// TIA Portal V18 export
DATA_BLOCK "Flowrate"   // DB205
{ S7_Optimized_Access := 'TRUE' }
VERSION : 0.1
// stored: AutoNumber true, DBAccessibleFromOPCUA true, IsOnlyStoredInLoadMemory false, IsRetainMemResEnabled false, IsWriteProtectedInAS false, MemoryReserve 100
   VAR
      Current : Struct
         "A" : Real;
         "B" : Real;
         Mixed : Real;
      END_STRUCT;
      "current in ml/min" : Struct
         "A" : Real;
         "B" : Real;
         Mixed : Real;
      END_STRUCT;
      "current in L/min" : Struct
         "A" : Real;
         "B" : Real;
         Mixed : Real;
      END_STRUCT;
      "current in KG/min" : Struct
         "A" : Real;
         "B" : Real;
         Mixed : Real;
      END_STRUCT;
      "Volume in ml" : Struct
         "A" : Real;
         "B" : Real;
         mixed : Real;
      END_STRUCT;
      "Volume in L" : Struct
         "A" : Real;
         "B" : Real;
         mixed : Real;
      END_STRUCT;
      "Volume in Kg" : Struct
         "A" : Real;
         "B" : Real;
         mixed : Real;
      END_STRUCT;
      "Current Volume" : Struct
         "A" : Real;
         "B" : Real;
         mixed : Real;
      END_STRUCT;
      "Current Flowrate" : Struct
         "A" : Real;
         "B" : Real;
         mixed : Real;
      END_STRUCT;
   END_VAR
   VAR RETAIN
      "selection ml/lit/kg" : Int := 1;
   END_VAR
   VAR
      Selected : Struct
         ml : Bool;
         cm3 : Bool;
         litre : Bool;
         kg : Bool;
         g { ExternalAccessible := 'False'; ExternalVisible := 'False'; ExternalWritable := 'False'} : Bool;
      END_STRUCT;
      tolerence : Struct
         Mixed : Real;
         Percentage : Real;
         "Mixed +" : Real;
         "Mixed -" : Real;
         Error : Bool;
      END_STRUCT;
      "current in g/min" : Struct
         "A" : Real;
         "B" : Real;
         Mixed : Real;
      END_STRUCT;
      "Volume in g" : Struct
         "A" : Real;
         "B" : Real;
         mixed : Real;
      END_STRUCT;
   END_VAR
BEGIN
END_DATA_BLOCK
